Universal Robots PolyScope program: rtde_control_CENSE.urp

Program rtde_control_CENSE (createdIn=3.2.19275.0 lastSavedIn=3.3.3.292 directory=/programs/usbdisk installation=rtde_installation_1 robotSerialNumber=2016353342)
Calibrated DH parameters: a=[0.000267, -0.004968, -0.38579, -0.000031, 0.00014, 0]; d=[0.089344, 354.021734, -340.399194, -13.511785, 0.094893, 0.082656]; alpha=[1.570332, -0.001201, 0.005165, 1.570021, -1.570286, 0]; deltaTheta=[0.000075, -1.559103, 1.739545, -0.180319, -0.000106, -0.000018]
BeforeStart
  tmp := p[0,0,0,0,0,0]
  Script: write_output_integer_register(0, 0)
  setp := Joint_6_name
  setj := get_actual_joint_positions()
  Script: rtde_set_watchdog("input_int_register_0", 1, "PAUSE")
  Script: sync()
Robot Program (runOnlyOnce=false motionType=MoveJ speed=1.047198 acceleration=1.396263 recalculateMotions=false)
  Script: sync()
  Script: write_output_integer_register(1,0)
  If read_input_integer_register(1)≟1
    Script: write_output_integer_register(1,1)
    MoveJ speed 60 deg/s, acceleration 80 deg/s^2 (recalculateMotions=false)
      Waypoint Wegpunkt (Variable): variable=setj
  Else 
    MoveL speed 250 mm/s, acceleration 1200 mm/s^2 (recalculateMotions=true) tcp=TCP; feature=Base
      Waypoint Waypoint (Variable): variable=setp
  Script: write_output_integer_register(1,0)
  Script: write_output_integer_register(0, 1)
Thread Thread_1 (runOnlyOnce=false trackProgramExecution=false)
  Loop Forever
    Script: sync()
    tmp := p[0,0,0,0,0,0]
    setp := get_actual_tcp_pose()
    setj := get_actual_joint_positions()
    Script: tmp[0] = read_input_float_register(0)
    Script: tmp[1] = read_input_float_register(1)
    Script: tmp[2] = read_input_float_register(2)
    Script: tmp[3] = read_input_float_register(3)
    Script: tmp[4] = read_input_float_register(4)
    Script: tmp[5] = read_input_float_register(5)
    If tmp != p[0,0,0,0,0,0]
      If read_input_integer_register(1)≟1
        setj := [tmp[0],tmp[1],tmp[2],tmp[3],tmp[4],tmp[5]]
      Else 
        setp := tmp
    Script: sync()
